// TIA Portal project "Selecao_peca" (V11)

(* hardware
DEVICE "S7300/ET200M station_1"  SIMATIC 300-Station
   slot 0: "Rail_0"  Rail  6ES7 390-1***0-0AA0
   slot 1: "PS 307 5A_1"  PS 307 5A  6ES7 307-1EA01-0AA0
   slot 2: "PLC_1"  CPU 314C-2 PN/DP  6ES7 314-6EH04-0AB0  V3.3
      slot 2: "PROFINET interface_1"  PN-IO
         slot 1: "Port_1"  Port
         slot 2: "Port_2"  Port
      slot 5: "DI24/DO16_1"  DI24/DO16
      slot 6: "AI5/AO2_1"  AI5/AO2
      slot 7: "Count_1"  Counter
      slot 8: "Positioning_1"  Positioning
   slot 4: "DI32 x 24VDC_1"  DI32xDC24V  6ES7 321-1BL00-0AA0
   slot 5: "DO16 x 24VDC / 0.5A_1"  DO16xDC24V/0.5A  6ES7 322-1BH01-0AA0
*)

// ===== PLC "PLC_1"  CPU 314C-2 PN/DP =====

VAR_GLOBAL   // PLC tag table "Default tag table"
   "Modo auto" AT %I125.5 : Bool;
   "relay" AT %Q124.0 : Bool;
   "P0_begin" AT %M124.1 : Bool;   // LUGAR
   "P37_vquit" AT %M124.2 : Bool;   // LUGAR
   "P2_caixapreta1" AT %M124.3 : Bool;   // LUGAR
   "P3_caixapreta1stop" AT %M124.4 : Bool;   // LUGAR
   "P4_caixapreta2" AT %M124.5 : Bool;   // LUGAR
   "P5_caixapreta2stop" AT %M124.6 : Bool;   // LUGAR
   "P6_esteiraesq-Esteira2^-Esteira1v" AT %M124.7 : Bool;   // LUGAR
   "P7_P6_esteiraesqstop" AT %M125.0 : Bool;   // LUGAR
   "P8_esteiraparada" AT %M125.1 : Bool;   // LUGAR
   "P9_esteiraparadastop" AT %M125.2 : Bool;   // LUGAR
   "P10_feijoada" AT %M125.3 : Bool;   // LUGAR
   "P11_feijoadastop" AT %M125.4 : Bool;   // LUGAR
   "P12_Mag1/2A^" AT %M125.5 : Bool;   // LUGAR
   "P13_Mag1/2A^stop" AT %M125.6 : Bool;   // LUGAR
   "P14_Mag1/2A^-Mag1/2Fv" AT %M125.7 : Bool;   // LUGAR
   "P15_Mag1/2A^-Mag1/2Fvstop" AT %M126.0 : Bool;   // LUGAR
   "P16_Mag1/2Fv" AT %M126.1 : Bool;   // LUGAR
   "P17_Mag1/2Fvstop" AT %M126.2 : Bool;   // LUGAR
   "P18_Tempeca" AT %M126.3 : Bool;   // LUGAR
   "P19_Tempecastop" AT %M126.4 : Bool;   // LUGAR
   "P20_Esteira1/2v-profRv-profE^" AT %M126.5 : Bool;   // LUGAR
   "P21_P20stop" AT %M126.6 : Bool;   // LUGAR
   "P22_P20stop-profR^" AT %M126.7 : Bool;   // LUGAR
   "P23_Cimaigual1" AT %M127.0 : Bool;   // LUGAR
   "P24_P23stop" AT %M127.1 : Bool;   // LUGAR
   "P25_estendido-ProfEv-ProfR^" AT %M127.2 : Bool;   // LUGAR
   "P26_P25stop" AT %M127.3 : Bool;   // LUGAR
   "P27_ProfRv-Esteira1^" AT %M127.4 : Bool;   // LUGAR
   "P28_P27stop" AT %M127.5 : Bool;   // LUGAR
   "P29_indigual1" AT %M127.6 : Bool;   // LUGAR
   "P30_P29stop" AT %M127.7 : Bool;   // LUGAR
   "P31_roubado-Esteira1v-Esteira2^" AT %M128.0 : Bool;   // LUGAR
   "P32_P31stop" AT %M128.1 : Bool;   // LUGAR
   "P33_chegou-Esteira1v" AT %M128.2 : Bool;   // LUGAR
   "P34_P33stop" AT %M128.3 : Bool;   // LUGAR
   "P35_accomplished" AT %M128.4 : Bool;   // LUGAR
   "P36_P35stop" AT %M128.5 : Bool;   // LUGAR
   "T0_bstart" AT %M128.6 : Bool;   // TRANSICAO
   "T96_sempre" AT %M128.7 : Bool;   // TRANSICAO
   "T20_notvquit" AT %M129.1 : Bool;   // TRANSICAO
   "T94_notT48" AT %M129.2 : Bool;   // TRANSICAO
   "T3" AT %M129.5 : Bool;   // TRANSICAO
   "T4" AT %M129.6 : Bool;   // TRANSICAO
   "T5" AT %M129.7 : Bool;   // TRANSICAO
   "T6" AT %M130.0 : Bool;   // TRANSICAO
   "T7" AT %M130.1 : Bool;   // TRANSICAO
   "T8" AT %M130.2 : Bool;   // TRANSICAO
   "T9" AT %M130.3 : Bool;   // TRANSICAO
   "T10" AT %M130.4 : Bool;   // TRANSICAO
   "T11" AT %M130.5 : Bool;   // TRANSICAO
   "T12" AT %M130.6 : Bool;   // TRANSICAO
   "T13" AT %M130.7 : Bool;   // TRANSICAO
   "T14" AT %M131.0 : Bool;   // TRANSICAO
   "T15" AT %M131.1 : Bool;   // TRANSICAO
   "T16" AT %M131.2 : Bool;   // TRANSICAO
   "T17" AT %M131.3 : Bool;   // TRANSICAO
   "T18" AT %M131.4 : Bool;   // TRANSICAO
   "T19" AT %M131.5 : Bool;   // TRANSICAO
   "T21" AT %M131.7 : Bool;   // TRANSICAO
   "T22" AT %M132.0 : Bool;   // TRANSICAO
   "T23" AT %M132.1 : Bool;   // TRANSICAO
   "T24" AT %M132.2 : Bool;   // TRANSICAO
   "T25" AT %M132.3 : Bool;   // TRANSICAO
   "T26" AT %M132.4 : Bool;   // TRANSICAO
   "T27" AT %M132.5 : Bool;   // TRANSICAO
   "T28" AT %M132.6 : Bool;   // TRANSICAO
   "T29" AT %M132.7 : Bool;   // TRANSICAO
   "T30" AT %M133.0 : Bool;   // TRANSICAO
   "T31" AT %M133.1 : Bool;   // TRANSICAO
   "T32" AT %M133.2 : Bool;   // TRANSICAO
   "T33" AT %M133.3 : Bool;   // TRANSICAO
   "T34" AT %M133.4 : Bool;   // TRANSICAO
   "T35" AT %M133.5 : Bool;   // TRANSICAO
   "T36" AT %M133.6 : Bool;   // TRANSICAO
   "T37" AT %M133.7 : Bool;   // TRANSICAO
   "T38" AT %M134.0 : Bool;   // TRANSICAO
   "T39" AT %M134.1 : Bool;   // TRANSICAO
   "T40" AT %M134.2 : Bool;   // TRANSICAO
   "T41" AT %M134.3 : Bool;   // TRANSICAO
   "T42" AT %M134.4 : Bool;   // TRANSICAO
   "T43" AT %M134.5 : Bool;   // TRANSICAO
   "T44" AT %M134.6 : Bool;   // TRANSICAO
   "T45" AT %M134.7 : Bool;   // TRANSICAO
   "T46" AT %M135.0 : Bool;   // TRANSICAO
   "T47" AT %M135.1 : Bool;   // TRANSICAO
   "T48" AT %M135.2 : Bool;   // TRANSICAO
   "T49" AT %M135.3 : Bool;   // TRANSICAO
   "T50" AT %M135.4 : Bool;   // TRANSICAO
   "T51" AT %M135.5 : Bool;   // TRANSICAO
   "T52" AT %M135.6 : Bool;   // TRANSICAO
   "T53" AT %M135.7 : Bool;   // TRANSICAO
   "T54" AT %M136.0 : Bool;   // TRANSICAO
   "T55" AT %M136.1 : Bool;   // TRANSICAO
   "T56" AT %M136.2 : Bool;   // TRANSICAO
   "T57" AT %M136.3 : Bool;   // TRANSICAO
   "T58" AT %M136.4 : Bool;   // TRANSICAO
   "T59" AT %M136.5 : Bool;   // TRANSICAO
   "T60" AT %M136.6 : Bool;   // TRANSICAO
   "T61" AT %M136.7 : Bool;   // TRANSICAO
   "T62" AT %M137.0 : Bool;   // TRANSICAO
   "T63" AT %M137.1 : Bool;   // TRANSICAO
   "T64" AT %M137.2 : Bool;   // TRANSICAO
   "T65" AT %M137.3 : Bool;   // TRANSICAO
   "T66" AT %M137.4 : Bool;   // TRANSICAO
   "T67" AT %M137.5 : Bool;   // TRANSICAO
   "T68" AT %M137.6 : Bool;   // TRANSICAO
   "T69" AT %M137.7 : Bool;   // TRANSICAO
   "T70" AT %M138.0 : Bool;   // TRANSICAO
   "T71" AT %M138.1 : Bool;   // TRANSICAO
   "T72" AT %M138.2 : Bool;   // TRANSICAO
   "T73" AT %M138.3 : Bool;   // TRANSICAO
   "T74" AT %M138.4 : Bool;   // TRANSICAO
   "T75" AT %M138.5 : Bool;   // TRANSICAO
   "T76" AT %M138.6 : Bool;   // TRANSICAO
   "T77" AT %M138.7 : Bool;   // TRANSICAO
   "T78" AT %M139.0 : Bool;   // TRANSICAO
   "T79" AT %M139.1 : Bool;   // TRANSICAO
   "T80" AT %M139.2 : Bool;   // TRANSICAO
   "T81" AT %M139.3 : Bool;   // TRANSICAO
   "T82" AT %M139.4 : Bool;   // TRANSICAO
   "T83" AT %M139.5 : Bool;   // TRANSICAO
   "T84" AT %M139.6 : Bool;   // TRANSICAO
   "T85" AT %M139.7 : Bool;   // TRANSICAO
   "T86" AT %M140.0 : Bool;   // TRANSICAO
   "T87" AT %M140.1 : Bool;   // TRANSICAO
   "T88" AT %M140.2 : Bool;   // TRANSICAO
   "T89" AT %M140.3 : Bool;   // TRANSICAO
   "T90" AT %M140.4 : Bool;   // TRANSICAO
   "T91" AT %M140.5 : Bool;   // TRANSICAO
   "T92" AT %M140.6 : Bool;   // TRANSICAO
   "T93" AT %M140.7 : Bool;   // TRANSICAO
   "T95" AT %M141.1 : Bool;   // TRANSICAO
   "T97" AT %M141.3 : Bool;   // TRANSICAO
   "T98" AT %M141.4 : Bool;   // TRANSICAO
   "T99" AT %M141.5 : Bool;   // TRANSICAO
   "T100" AT %M141.6 : Bool;   // TRANSICAO
   "T101" AT %M141.7 : Bool;   // TRANSICAO
   "T102" AT %M142.0 : Bool;   // TRANSICAO
   "T103" AT %M142.1 : Bool;   // TRANSICAO
   "T104" AT %M142.2 : Bool;   // TRANSICAO
   "T105" AT %M142.3 : Bool;   // TRANSICAO
   "T106" AT %M142.4 : Bool;   // TRANSICAO
   "T107" AT %M142.5 : Bool;   // TRANSICAO
   "T108" AT %M142.6 : Bool;   // TRANSICAO
   "T109" AT %M142.7 : Bool;   // TRANSICAO
   "T110" AT %M143.0 : Bool;   // TRANSICAO
   "T111" AT %M143.1 : Bool;   // TRANSICAO
   "T112" AT %M143.2 : Bool;   // TRANSICAO
   "T113" AT %M143.3 : Bool;   // TRANSICAO
   "T114" AT %M143.4 : Bool;   // TRANSICAO
   "T115" AT %M143.5 : Bool;   // TRANSICAO
   "Start" AT %I125.4 : Bool;
   "Stop" AT %I125.3 : Bool;
   "Quit" AT %I125.2 : Bool;
   "Mag1A" AT %Q4.5 : Bool;
   "Mag2A" AT %Q4.7 : Bool;
   "Mag1F" AT %Q4.4 : Bool;
   "Mag2F" AT %Q4.6 : Bool;
   "FCMag1" AT %I0.7 : Bool;
   "FCMag2" AT %I1.2 : Bool;
   "Smag1A" AT %I0.5 : Bool;
   "Smag1F" AT %I0.6 : Bool;
   "Smag2A" AT %I1.0 : Bool;
   "Smag2F" AT %I1.1 : Bool;
   "Esteira1" AT %Q4.0 : Bool;
   "Esteira2" AT %Q4.1 : Bool;
   "Scapac" AT %I0.1 : Bool;
   "ProfE" AT %Q4.2 : Bool;
   "ProfR" AT %Q4.3 : Bool;
   "Sprof" AT %I0.2 : Bool;
   "Sindut" AT %I0.4 : Bool;
   "SoticBarreir" AT %I0.0 : Bool;
   "Cima" AT %M143.6 : Bool;   // VARIAVEIS
   "Ind" AT %M143.7 : Bool;   // VARIAVEIS
   "blocos" AT %MW144 : Int;   // VARIAVEIS
   "vquit" AT %M146.0 : Bool;   // VARIAVEIS
   "Verde" AT %Q124.4 : Bool;
   "Vermelho" AT %Q124.5 : Bool;
   "Azul" AT %Q124.6 : Bool;
   "Inicializadora" AT %M129.0 : Bool;
   "vstart" AT %M146.1 : Bool;   // VARIAVEIS
END_VAR

ORGANIZATION_BLOCK "Main"   // OB1, LAD
TITLE = "Main Program Sweep (Cycle)"
{ S7_Optimized_Access := 'FALSE' }
VERSION : 0.1
   VAR_TEMP
      OB1_EV_CLASS : Byte;   // Bits 0-3 = 1 (Coming event), Bits 4-7 = 1 (Event class 1)
      OB1_SCAN_1 : Byte;   // 1 (Cold restart scan 1 of OB 1), 3 (Scan 2-n of OB 1)
      OB1_PRIORITY : Byte;   // Priority of OB Execution
      OB1_OB_NUMBR : Byte;   // 1 (Organization block 1, OB1)
      OB1_RESERVED_1 : Byte;   // Reserved for system
      OB1_RESERVED_2 : Byte;   // Reserved for system
      OB1_PREV_CYCLE : Int;   // Cycle time of previous OB1 scan (milliseconds)
      OB1_MIN_CYCLE : Int;   // Minimum cycle time of OB1 (milliseconds)
      OB1_MAX_CYCLE : Int;   // Maximum cycle time of OB1 (milliseconds)
      OB1_DATE_TIME : Date_And_Time;   // Date and time OB1 started
   END_VAR
BEGIN
END_ORGANIZATION_BLOCK